# EPICS substitutions: db/Beckhoff_MX/ecmcMO7221-9016-CSP.substitutions
#- CSP drive and encoder records for MO7221-9016 safety drives.
file "ecmcEL72XX_DRV_CSP.template" {
  pattern { CH_ID }
    { 01 }
}

file "ecmcEL72XX_ENC.template" {
  pattern { CH_ID }
    { 01 }
}

file "ecmcMO7221-9016.template" {
  pattern { CH_ID }
    { 01 }
}

file "ecmc_analogInput-chX.template" {
  pattern { CH_ID, sourceName, KEY, suffix, DESC, EGU, ESLO, PREC, LOPR, HOPR, LOLO, LOW, HIGH, HIHI, HYST, LLSV, LSV, HSV, HHSV }
    { 01, "velocityActual", "Drv", "-VelAct", "Actual Vel", "rad/s", 2.3406E-5, 3, 0, 0, 0, 0, 0, 0, 0, "NO_ALARM", "NO_ALARM", "NO_ALARM", "NO_ALARM" }
    { 01, "torqueActual", "Drv", "-TrqAct", "Actual Trq", "%", 0.1, 1, -100, 100, 0, -80, 80, 0, 0, "NO_ALARM", "NO_ALARM", "MINOR", "NO_ALARM" }
    { 01, "voltageActual", "Drv", "-VolAct", "Actual Voltage", "V", 0.001, 3, 0, 60, 8, 20, 49, 50, 0.25, "MAJOR", "MINOR", "MINOR", "MAJOR" }
    { 01, "temperatureActual", "Drv", "-TmpAct", "PCB Temperature", "degC", 0.1, 1, -40, 150, 0, 0, 0, 0, 0, "NO_ALARM", "NO_ALARM", "NO_ALARM", "NO_ALARM" }
}

file "ecmc_binaryOutput-chX.template" {
  pattern { CH_ID, sourceName, KEY, DESC, ZNAM, ONAM }
    { "", "binaryOutput01", "Rst", "Reset safety application", "Idle", "Reset" }
    { "", "binaryOutput02", "Run", "Run safety application", "Stopped", "Run" }
}

file "ecmc_binaryInput-chX.template" {
  pattern { CH_ID, sourceName, KEY, DESC }
    { "", "binaryInput01", "ComErr", "Communication error" }
    { "", "binaryInput02", "ComStartup", "Communication startup" }
    { "", "binaryInput03", "FBDeactive", "Function block deactivated" }
    { "", "binaryInput04", "FBErr", "Function block error" }
    { "", "binaryInput05", "FBRun", "Function block running" }
    { "", "binaryInput06", "InRun", "Input running" }
    { "", "binaryInput07", "OtherErr", "Other error" }
    { "", "binaryInput08", "ReduceSpeed", "Reduced speed active" }
}

file "ecmc_controlWord-chX.template" {
  pattern { CH_ID, KEY, sourceName }
    { 01, FSoE-CmdOut, fsoe_cmd_out_ }
    { 01, FSoE-DataOut, fsoe_data_out_ }
    { 01, FSoE-CrcOut, fsoe_crc_out_ }
    { 01, FSoE-ConnIdOut, fsoe_conn_id_out_ }
}

file "ecmc_status-chX.template" {
  pattern { CH_ID, KEY, sourceName, suffix }
    { 01, FSoE-CmdIn, fsoe_cmd_in_, "" }
    { 01, FSoE-DataIn, fsoe_data_in_, "" }
    { 01, FSoE-CrcIn, fsoe_crc_in_, "" }
    { 01, FSoE-ConnIdIn, fsoe_conn_id_in_, "" }
    { 01, FSoE-StateIn, fsoe_state_in_, "" }
    { 01, FSoE-CycCntIn, fsoe_cycle_counter_in_, "" }
}
